(* PLC project prj, KAIST_DSLAB noNameNow 1, author bwkim *)
(* stored: creationDateTime 2015-9-6T01:13:23, modificationDateTime 2015-9-6T01:13:23 *)

PROGRAM Program1____CTU_and_TON
  VAR
    LEVEL_CTR : null;
  END_VAR
  VAR
    PULSE : null;
  END_VAR
  VAR_OUTPUT
    TON_et : INT;
  END_VAR
  VAR_IN_OUT
    CTU_UP : BOOL := FALSE;
  END_VAR

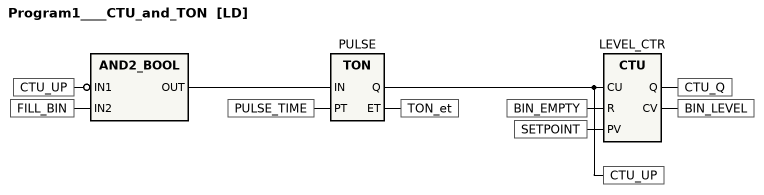
(* LD diagram, written out as Structured Text *)
PULSE(IN := AND2_BOOL(NOT CTU_UP, FILL_BIN), PT := PULSE_TIME);
CTU_UP := PULSE.Q;
LEVEL_CTR(CU := PULSE.Q, R := BIN_EMPTY, PV := SETPOINT);
CTU_Q := LEVEL_CTR.Q;
TON_et := PULSE.ET;
BIN_LEVEL := LEVEL_CTR.CV;
END_PROGRAM
